// TIA Portal project "Soru3" (V15)

(* hardware
DEVICE "S7-1200 station_1"  S7-1200 Station
   slot 0: "Rack_0"  S7-1200 Rack  Rack  V1.0
   slot 1: "PLC_1"  CPU 1214C DC/DC/DC  6ES7 214-1AG40-0XB0  V4.2
*)

// ===== PLC "PLC_1"  CPU 1214C DC/DC/DC =====

VAR_GLOBAL   // PLC tag table "Default tag table"
   "Durdur" AT %I0.0 : Bool;
   "Baslat" AT %I0.1 : Bool;
   "Sensor" AT %I0.2 : Bool;
   "Konveyor_1" AT %Q0.0 : Bool;
   "Konveyor_2" AT %Q0.1 : Bool;
END_VAR

// folder: System blocks/Program resources

DATA_BLOCK "IEC_Timer_0_DB"   // DB1
{ S7_Optimized_Access := 'TRUE' }
AUTHOR : Simatic
FAMILY : IEC
NAME : IEC_TMR
VERSION : 1.0
// stored: InstanceOfName IEC_TIMER
"IEC_TIMER"
BEGIN
END_DATA_BLOCK

DATA_BLOCK "IEC_Timer_0_DB_1"   // DB2
{ S7_Optimized_Access := 'TRUE' }
AUTHOR : Simatic
FAMILY : IEC
NAME : IEC_TMR
VERSION : 1.0
// stored: InstanceOfName IEC_TIMER
"IEC_TIMER"
BEGIN
END_DATA_BLOCK

DATA_BLOCK "IEC_Counter_0_DB"   // DB3
{ S7_Optimized_Access := 'TRUE' }
AUTHOR : Simatic
FAMILY : IEC
NAME : UCNTR
VERSION : 1.2
// stored: InstanceOfName IEC_UCOUNTER
"IEC_UCOUNTER"
BEGIN
END_DATA_BLOCK

// folder: (top level)

ORGANIZATION_BLOCK "Main"   // OB1, LAD, ProgramCycle
TITLE = "Main Program Sweep (Cycle)"
{ S7_Optimized_Access := 'TRUE' }
VERSION : 0.1
   VAR_INPUT
      Initial_Call : Bool;   // Initial call of this OB
      Remanence : Bool;   // =True, if remanent data are available
   END_VAR
BEGIN

REGION Network 1: Zaman dögüngüsü
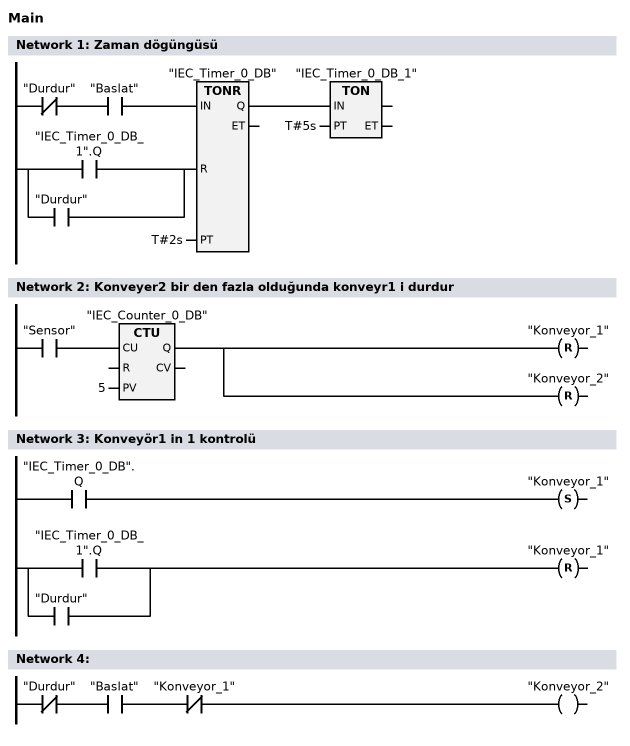
   "IEC_Timer_0_DB".TONR(IN := NOT "Durdur" AND "Baslat", R := "IEC_Timer_0_DB_1".Q OR "Durdur", PT := T#2s);
   "IEC_Timer_0_DB_1".TON(IN := "IEC_Timer_0_DB".Q, PT := T#5s);
END_REGION

REGION Network 2: Konveyer2 bir den fazla olduğunda konveyr1 i durdur
   "IEC_Counter_0_DB".CTU(CU := "Sensor", PV := 5);
   IF "IEC_Counter_0_DB".Q THEN
       "Konveyor_1" := FALSE;
       "Konveyor_2" := FALSE;
   END_IF;
END_REGION

REGION Network 3: Konveyör1 in 1 kontrolü
   RUNG wire#powerrail
      Contact( "IEC_Timer_0_DB".Q )
      S_Coil( "Konveyor_1" )
   END_RUNG
   RUNG wire#powerrail
      Contact( "IEC_Timer_0_DB_1".Q )
      wire#w1
      R_Coil( "Konveyor_1" )
   END_RUNG
   RUNG wire#powerrail
      Contact( "Durdur" )
   END_RUNG wire#w1
   // the same network as SCL:
   IF "IEC_Timer_0_DB".Q THEN "Konveyor_1" := TRUE; END_IF;
   IF "IEC_Timer_0_DB_1".Q OR "Durdur" THEN "Konveyor_1" := FALSE; END_IF;
END_REGION

REGION Network 4
   RUNG wire#powerrail
      I_Contact( "Durdur" )
      Contact( "Baslat" )
      I_Contact( "Konveyor_1" )
      Coil( "Konveyor_2" )
   END_RUNG
   // the same network as SCL:
   "Konveyor_2" := NOT "Durdur" AND "Baslat" AND NOT "Konveyor_1";
END_REGION
END_ORGANIZATION_BLOCK